// TIA Portal V16 export
// export: Created 2025-12-29T07:34:59.928153Z, ExportSetting WithDefaults, DisplayName Totally Integrated Automation Portal, DisplayVersion V16, DisplayName TIA Portal Version Control Interface, DisplayVersion V16, DisplayName TIA Portal Openness, DisplayVersion V16, DisplayName STEP 7 Professional, DisplayVersion V16, DisplayName STEP 7 Safety, DisplayVersion V16, DisplayName WinCC Professional, DisplayVersion V16
VAR_GLOBAL   // PLC tag table "Standard-Variablentabelle"
   Clock_Byte AT %MB0 : Byte;
   Clock_10Hz AT %M0.0 : Bool;
   Clock_5Hz AT %M0.1 : Bool;
   "Clock_2.5Hz" AT %M0.2 : Bool;
   Clock_2Hz AT %M0.3 : Bool;
   "Clock_1.25Hz" AT %M0.4 : Bool;
   Clock_1Hz AT %M0.5 : Bool;
   "Clock_0.625Hz" AT %M0.6 : Bool;
   "Clock_0.5Hz" AT %M0.7 : Bool;
   Status AT %MW2 : Int;
   Awaria_Potwierdzona AT %M1.0 : Bool;
   System_Pracuje AT %M1.1 : Bool;
   Reset_Potwierdzony AT %M1.2 : Bool;
   Awaria_Aktywna AT %M1.3 : Bool;
   state AT %MW4 : Int;
   Pamiec_Typ_4 AT %M1.4 : Bool;
   Pamiec_Typ_1 AT %M1.5 : Bool;
END_VAR
